(* CODESYS project untitled1.library
   Placeholder: TwinCAT_LIB
   Title: TwinCAT_LIB
   Version: 1.31
   Description: Baisc library's for s88 programming
   Company: Farnwood Engineering

Project tree, tasks and I/O mapping:
  libraries: Tc2_Standard, * (Beckhoff Automation GmbH); Tc2_System, * (Beckhoff Automation GmbH); Tc3_Module, * (Beckhoff Automation GmbH)
  DUTs/
  GVLs/
    POUs/
      LIB/
        1. Control Modules/
          1. DEV_Base/
            function block FB_DeviceBase [ST]
            data type stDevBase
          2. DEV_AnaIn/
            function block FB_DEV_AnaIn [ST]
            interface ITF_DEV_AnaIn
          3. DEV_DigIn/
            function block FB_DEV_DigIn [ST]: FB_init, Force, ResetForce, ActualValue, FallingEdge, RisingEdge
            interface ITF_DigIn: FB_init, Force, ResetForce, ActualValue, FallingEdge, RisingEdge
          4. DEV_Valve/
            ENUMs/
              data type E_ValveState
            STRUCTs/
              data type stDevValve
            function block DEV_Valve [ST]: _FExceptions, _StHmi, Close, Open, Reset, SetMode, ActualState, EmergencyStatus, OperatingMode
            interface ITF_Valve: Close, Open, Reset, SetMode, ActualState, EmergencyStatus, OperatingMode
          5. DEV_ControlValve/
            ENUMs/
              data type E_CtrlValveState
            STRUCTs/
            function block DEV_CtrlValve [ST]: EmergencyStatus, OperatingMode, OutputValue, Reset, SetMode, SetValue
            interface ITF_ControlValve: Reset, SetMode, SetValue, EmergencyStatus, OperatingMode, OutputValue
          6. DEV_Motor/
            ENUMs/
              data type E_MotorState
            STRUCTs/
            interface ITF_Motor: Auto, Manueel, Reset, Richting_L, Richting_R, Start, Stop, Toerental, ActualState, Error_State, State
          7. DEV_ControlMotor/
          ENUMs/
            data type E_OperationMode
          function block FB_Devices [ST]
        2. Equipment Modules/
          1. FB_Base/
            function block FB_EMbase [ST]
            data type stEMbase
          2. FB_Machine_PackML/
            data type E_State_PackML
            function block FB_Machine_PackML [ST]: Abort, Aborting_SC, Clear, Clearing_SC, Completing_SC, Execute_SC, Hold, Holding_SC, Reset, Resetting_SC, Start, Starting_SC, Stop, Stopping_SC, Suspend, Suspending_SC, Unhold, Unholding_SC, Unsuspend, Unsuspending_SC, State, FB_init
            interface ITF_PackML: Abort, Aborting_SC, Clear, Clearing_SC, Completing_SC, Execute_SC, Hold, Holding_SC, Reset, Resetting_SC, Start, Starting_SC, Stop, Stopping_SC, Suspend, Suspending_SC, Unhold, Unholding_SC, Unsuspend, Unsuspending_SC, State, FB_init
            data type STRUCT_fb_mem
          2. FB_Transport/
            data type E_Transport
            function block FB_Transport [ST]: Abort, Clear, Reset, Start, Stop, RPM, State, Tag
            interface ITF_FB_Transport: Abort, Clear, Reset, Start, Stop, RPM, State, Tag
            data type Str_FB_Transport
          3. FB_Transport_Mechanische_Stop/
            data type E_Mechanische_Stop
            function block FB_Mechanische_Stop [ST]: Close, Open, State, Tag
            interface ITF_FB_Transport_Mechanische_Stop: Close, Open, State, Tag
        3. Units/
          1. UN_Base/
            function block FB_UN_base [ST]
            data type stUNbase
        4. Management layer/
          FB_Alarmhandler/
      program MAIN [ST]
  Version/
    global variables Global_Version
  VISUs/
*)

// GVLs/POUs/LIB/1. Control Modules/1. DEV_Base/stDevBase
TYPE stDevBase :
STRUCT
	sTagName : STRING;
	sDescription : STRING;
END_STRUCT
END_TYPE

// GVLs/POUs/LIB/1. Control Modules/4. DEV_Valve/ENUMs/E_ValveState
{attribute 'qualified_only'}
{attribute 'strict'}
TYPE E_ValveState :
(
	Unknown := 0,
	Open := 1,
	Closed := 2,
	Opening := 3,
	Closing := 4,
	Error := -1
);
END_TYPE

// GVLs/POUs/LIB/1. Control Modules/4. DEV_Valve/STRUCTs/stDevValve
TYPE stDevValve :
STRUCT
	//Input to HMI
	bGetHmiError : BOOL;  //True = error
	bGetHmiStatus : BOOL; //True = Open || False = Closed
	eGetState : E_ValveState;
	eGetMode : E_OperationMode;
	
	//Output from HMI
	eSetMode : E_OperationMode; 
END_STRUCT
END_TYPE

// GVLs/POUs/LIB/1. Control Modules/5. DEV_ControlValve/ENUMs/E_CtrlValveState
{attribute 'qualified_only'}
{attribute 'strict'}
TYPE E_CtrlValveState :
(
	Unknown := 0,
	InPosition := 1,
	Moving := 2,
	Error := -1
);
END_TYPE

// GVLs/POUs/LIB/1. Control Modules/6. DEV_Motor/ENUMs/E_MotorState
{attribute 'qualified_only'}
{attribute 'strict'}
TYPE E_MotorState :
(
	Unknown := 0,
	Running := 1,
	Stalled := 2,
	SpeedingUp := 3,
	SpeedingDown := 4,
	Error := -1
);
END_TYPE

// GVLs/POUs/LIB/1. Control Modules/ENUMs/E_OperationMode
{attribute 'qualified_only'}
{attribute 'strict'}
TYPE E_OperationMode :
(
	Off := 0,
	Manual := 1,
	Automatic := 2
);
END_TYPE

// GVLs/POUs/LIB/2. Equipment Modules/1. FB_Base/stEMbase
TYPE stEMbase :
STRUCT
	sTagName : STRING;
	sDescription : STRING;
END_STRUCT
END_TYPE

// GVLs/POUs/LIB/2. Equipment Modules/2. FB_Machine_PackML/E_State_PackML
{attribute 'qualified_only'}
{attribute 'strict'}
TYPE E_State_PackML :
(
	IDLE	:= 0,
	STARTING,
	EXECUTE,
	COMPLETING,
	COMPLETE,
	RESETTING,
	HOLDING,
	HELD,
	UNHOLDING,
	SUSPENDING,
	SUSPENDED,
	UNSUSPENDING,
	ABORTING,
	ABORTED,
	CLEARING,
	STOPPING,
	STOPPED
);
END_TYPE

// GVLs/POUs/LIB/2. Equipment Modules/2. FB_Machine_PackML/STRUCT_fb_mem
TYPE STRUCT_fb_mem :
STRUCT
	//Properties
	State 			: E_State_PackML;
	//Methods
   	Abort 			: BOOL;
	Aborting_SC 	: BOOL;
	Clear 			: BOOL;
	Clearing_SC 	: BOOL;
	Execute_SC 		: BOOL;
	Completing_SC	: BOOL;
	Hold 			: BOOL;
	Holding_SC 		: BOOL;
	Reset 			: BOOL;
	Resetting_SC 	: BOOL;
	Start 			: BOOL;
	Starting_SC 	: BOOL;
	Stop 			: BOOL;
	Stopping_SC 	: BOOL;
	Suspend 		: BOOL;
	Suspending_SC 	: BOOL;
	Unhold 			: BOOL;
	Unholding_SC 	: BOOL;
	Unsuspend 		: BOOL;
	Unsuspending_SC : BOOL;
END_STRUCT
END_TYPE

// GVLs/POUs/LIB/2. Equipment Modules/2. FB_Transport/E_Transport
{attribute 'qualified_only'}
{attribute 'strict'}
TYPE E_Transport :
(
	IDLE := 0,
	STARTING,
	EXECUTE,
	STOPPING,
	STOPPED,
	ABORTING,
	ABORT,
	CLEARING,
	CLEARED,
	RESETTING
	
);
END_TYPE

// GVLs/POUs/LIB/2. Equipment Modules/2. FB_Transport/Str_FB_Transport
{attribute 'qualified_only'}
{attribute 'strict'}
TYPE Str_FB_Transport :
(
	enum_member := 0
);
END_TYPE

// GVLs/POUs/LIB/2. Equipment Modules/3. FB_Transport_Mechanische_Stop/E_Mechanische_Stop
{attribute 'qualified_only'}
{attribute 'strict'}
TYPE E_Mechanische_Stop :
(
	enum_member := 0
);
END_TYPE

// GVLs/POUs/LIB/3. Units/1. UN_Base/stUNbase
TYPE stUNbase :
STRUCT
	sTagName : STRING;
	sDescription : STRING;
END_STRUCT
END_TYPE

// Version/Global_Version
{attribute 'TcGenerated'}
{attribute 'no-analysis'}
{attribute 'linkalways'}
// This function has been automatically generated from the project information.
VAR_GLOBAL CONSTANT
	{attribute 'const_non_replaced'}
	stLibVersion_TwinCAT_LIB : ST_LibVersion := (iMajor := 1, iMinor := 31, iBuild := 0, iRevision := 0, nFlags := 1, sVersion := '1.31');
END_VAR

// GVLs/POUs/LIB/1. Control Modules/1. DEV_Base/FB_DeviceBase
FUNCTION_BLOCK FB_DeviceBase
VAR
	TagName : STRING;
	Description : STRING;
	TagID : INT;
END_VAR

END_FUNCTION_BLOCK

// GVLs/POUs/LIB/1. Control Modules/2. DEV_AnaIn/FB_DEV_AnaIn
FUNCTION_BLOCK FB_DEV_AnaIn EXTENDS FB_DeviceBase IMPLEMENTS ITF_DEV_AnaIn
VAR_INPUT
END_VAR
VAR_OUTPUT
END_VAR
VAR
END_VAR

END_FUNCTION_BLOCK

// GVLs/POUs/LIB/1. Control Modules/2. DEV_AnaIn/ITF_DEV_AnaIn
INTERFACE ITF_DEV_AnaIn

END_INTERFACE

// GVLs/POUs/LIB/1. Control Modules/3. DEV_DigIn/FB_DEV_DigIn
FUNCTION_BLOCK FB_DEV_DigIn EXTENDS FB_DeviceBase IMPLEMENTS ITF_DigIn
VAR
	
END_VAR

{warning 'add method implementation '}
METHOD FB_init : BOOL
VAR_INPUT
	(* if TRUE, the retain variables are initialized (warm start / cold start)*)
	bInitRetains	: BOOL;
	(* if TRUE, the instance afterwards gets moved into the copy code (online change)*)
	bInCopyCode	: BOOL;
END_VAR
END_METHOD

{warning 'add method implementation '}
METHOD Force : BOOL
VAR_INPUT
	ForceValue	: BOOL;
END_VAR
END_METHOD

{warning 'add method implementation '}
METHOD ResetForce : BOOL
END_METHOD

{warning 'add property implementation'}
PROPERTY ActualValue : BOOL
GET
END_GET
SET
END_SET
END_PROPERTY

{warning 'add property implementation'}
PROPERTY FallingEdge : BOOL
GET
END_GET
SET
END_SET
END_PROPERTY

{warning 'add property implementation'}
PROPERTY RisingEdge : BOOL
GET
END_GET
SET
END_SET
END_PROPERTY

END_FUNCTION_BLOCK

// GVLs/POUs/LIB/1. Control Modules/3. DEV_DigIn/ITF_DigIn
INTERFACE ITF_DigIn

METHOD FB_init : BOOL
VAR_INPUT
	bInitRetains : BOOL; // if TRUE, the retain variables are initialized (warm start / cold start)
	bInCopyCode : BOOL;  // if TRUE, the instance afterwards gets moved into the copy code (online change)
END_VAR
END_METHOD

METHOD Force : BOOL
VAR_INPUT
	ForceValue : BOOL;
END_VAR
END_METHOD

METHOD ResetForce : BOOL
VAR_INPUT
END_VAR
END_METHOD

PROPERTY ActualValue : BOOL
GET
END_GET
SET
END_SET
END_PROPERTY

PROPERTY FallingEdge : BOOL
GET
END_GET
SET
END_SET
END_PROPERTY

PROPERTY RisingEdge : BOOL
GET
END_GET
SET
END_SET
END_PROPERTY

END_INTERFACE

// GVLs/POUs/LIB/1. Control Modules/4. DEV_Valve/DEV_Valve
FUNCTION_BLOCK DEV_Valve EXTENDS FB_DeviceBase IMPLEMENTS ITF_Valve

VAR
	I_FeedbackOpen		AT	%I* : BOOL;
	I_FeedbackClosed 	AT 	%I* : BOOL;
	I_Estop				AT	%I*	: BOOL;
	Q_ValveOutput		AT	%Q*	: BOOL;
	
	s_eActualState				: E_ValveState;
	s_eOperatingMode			: E_OperationMode;
	s_tonFeedbackTime			: TON;
	
	bFeedbackError		: BOOL;
	bEstopActive		: BOOL;
	bBothFeedback		: BOOL;
END_VAR

METHOD _FExceptions : BOOL
VAR_INPUT
END_VAR
END_METHOD

METHOD PRIVATE _StHmi
VAR_INPUT
	stHMI : stDevValve;
END_VAR
END_METHOD

{warning 'add method implementation '}
METHOD Close : BOOL
END_METHOD

{warning 'add method implementation '}
METHOD Open : BOOL
END_METHOD

{warning 'add method implementation '}
METHOD Reset : BOOL
END_METHOD

{warning 'add method implementation '}
METHOD SetMode : BOOL
END_METHOD

{warning 'add property implementation'}
PROPERTY ActualState : E_ValveState
GET
END_GET
END_PROPERTY

{warning 'add property implementation'}
PROPERTY EmergencyStatus : BOOL
GET
END_GET
END_PROPERTY

{warning 'add property implementation'}
PROPERTY OperatingMode : BOOL
GET
END_GET
END_PROPERTY

END_FUNCTION_BLOCK

// GVLs/POUs/LIB/1. Control Modules/4. DEV_Valve/ITF_Valve
INTERFACE ITF_Valve

METHOD Close : BOOL
VAR_INPUT
END_VAR
END_METHOD

METHOD Open : BOOL
VAR_INPUT
END_VAR
END_METHOD

METHOD Reset : BOOL
VAR_INPUT
END_VAR
END_METHOD

METHOD SetMode : BOOL
VAR_INPUT
END_VAR
END_METHOD

PROPERTY ActualState : E_ValveState
GET
END_GET
END_PROPERTY

PROPERTY EmergencyStatus : BOOL
GET
END_GET
END_PROPERTY

PROPERTY OperatingMode : BOOL
GET
END_GET
END_PROPERTY

END_INTERFACE

// GVLs/POUs/LIB/1. Control Modules/5. DEV_ControlValve/DEV_CtrlValve
FUNCTION_BLOCK DEV_CtrlValve EXTENDS FB_DeviceBase IMPLEMENTS ITF_ControlValve
VAR_INPUT
END_VAR
VAR_OUTPUT
END_VAR
VAR
END_VAR

{warning 'add property implementation'}
PROPERTY EmergencyStatus : BOOL
GET
END_GET
END_PROPERTY

{warning 'add property implementation'}
PROPERTY OperatingMode : BOOL
GET
END_GET
END_PROPERTY

{warning 'add property implementation'}
PROPERTY OutputValue : REAL
GET
END_GET
END_PROPERTY

{warning 'add method implementation '}
METHOD Reset : BOOL
END_METHOD

{warning 'add method implementation '}
METHOD SetMode : BOOL
END_METHOD

{warning 'add method implementation '}
METHOD SetValue : BOOL
END_METHOD

END_FUNCTION_BLOCK

// GVLs/POUs/LIB/1. Control Modules/5. DEV_ControlValve/ITF_ControlValve
INTERFACE ITF_ControlValve

METHOD Reset : BOOL
VAR_INPUT
END_VAR
END_METHOD

METHOD SetMode : BOOL
VAR_INPUT
END_VAR
END_METHOD

METHOD SetValue : BOOL
VAR_INPUT
END_VAR
END_METHOD

PROPERTY EmergencyStatus : BOOL
GET
END_GET
END_PROPERTY

PROPERTY OperatingMode : BOOL
GET
END_GET
END_PROPERTY

PROPERTY OutputValue : REAL
GET
END_GET
END_PROPERTY

END_INTERFACE

// GVLs/POUs/LIB/1. Control Modules/6. DEV_Motor/ITF_Motor
INTERFACE ITF_Motor

METHOD Auto : BOOL
VAR_INPUT
END_VAR
END_METHOD

METHOD Manueel : BOOL
VAR_INPUT
END_VAR
END_METHOD

METHOD Reset : BOOL
VAR_INPUT
END_VAR
END_METHOD

METHOD Richting_L : BOOL
VAR_INPUT
END_VAR
END_METHOD

METHOD Richting_R : BOOL
VAR_INPUT
END_VAR
END_METHOD

METHOD Start : BOOL
VAR_INPUT
END_VAR
END_METHOD

METHOD Stop : BOOL
VAR_INPUT
END_VAR
END_METHOD

METHOD Toerental : INT
VAR_INPUT
END_VAR
END_METHOD

PROPERTY ActualState : BOOL
GET
END_GET
END_PROPERTY

PROPERTY Error_State : BOOL
GET
END_GET
END_PROPERTY

PROPERTY State : E_MotorState
GET
END_GET
END_PROPERTY

END_INTERFACE

// GVLs/POUs/LIB/1. Control Modules/FB_Devices
FUNCTION_BLOCK FB_Devices
VAR
	devValveV2012 : DEV_Valve := (TagName := 'V2012', Description := 'Standard Valve', TagID := 1);
	devValveV2020 : DEV_Valve := (TagName := 'V2020', Description := 'Standard Valve', TagID := 2);
	devValveV2021 : DEV_Valve := (TagName := 'V2021', Description := 'Standard Valve', TagID := 3);
	devValveV2022 : DEV_Valve := (TagName := 'V2022', Description := 'Standard Valve', TagID := 4);
END_VAR

devValveV2012();
devValveV2020();
devValveV2021();
devValveV2020();

END_FUNCTION_BLOCK

// GVLs/POUs/LIB/2. Equipment Modules/1. FB_Base/FB_EMbase
FUNCTION_BLOCK FB_EMbase
VAR
	TagName : STRING;
	Description : STRING;
	TagID : INT;
END_VAR

END_FUNCTION_BLOCK

// GVLs/POUs/LIB/2. Equipment Modules/2. FB_Machine_PackML/FB_Machine_PackML
FUNCTION_BLOCK FB_Machine_PackML IMPLEMENTS ITF_PackML
VAR
	fb_mem : STRUCT_fb_mem;
END_VAR

(*
$$$$$$$$\                                                                   $$\       $$$$$$$$\                     $$\                                         $$\                     
$$  _____|                                                                  $$ |      $$  _____|                    \__|                                        \__|                    
$$ |   $$$$$$\   $$$$$$\  $$$$$$$\  $$\  $$\  $$\  $$$$$$\   $$$$$$\   $$$$$$$ |      $$ |      $$$$$$$\   $$$$$$\  $$\ $$$$$$$\   $$$$$$\   $$$$$$\   $$$$$$\  $$\ $$$$$$$\   $$$$$$\  
$$$$$\ \____$$\ $$  __$$\ $$  __$$\ $$ | $$ | $$ |$$  __$$\ $$  __$$\ $$  __$$ |      $$$$$\    $$  __$$\ $$  __$$\ $$ |$$  __$$\ $$  __$$\ $$  __$$\ $$  __$$\ $$ |$$  __$$\ $$  __$$\ 
$$  __|$$$$$$$ |$$ |  \__|$$ |  $$ |$$ | $$ | $$ |$$ /  $$ |$$ /  $$ |$$ /  $$ |      $$  __|   $$ |  $$ |$$ /  $$ |$$ |$$ |  $$ |$$$$$$$$ |$$$$$$$$ |$$ |  \__|$$ |$$ |  $$ |$$ /  $$ |
$$ |  $$  __$$ |$$ |      $$ |  $$ |$$ | $$ | $$ |$$ |  $$ |$$ |  $$ |$$ |  $$ |      $$ |      $$ |  $$ |$$ |  $$ |$$ |$$ |  $$ |$$   ____|$$   ____|$$ |      $$ |$$ |  $$ |$$ |  $$ |
$$ |  \$$$$$$$ |$$ |      $$ |  $$ |\$$$$$\$$$$  |\$$$$$$  |\$$$$$$  |\$$$$$$$ |      $$$$$$$$\ $$ |  $$ |\$$$$$$$ |$$ |$$ |  $$ |\$$$$$$$\ \$$$$$$$\ $$ |      $$ |$$ |  $$ |\$$$$$$$ |
\__|   \_______|\__|      \__|  \__| \_____\____/  \______/  \______/  \_______|      \________|\__|  \__| \____$$ |\__|\__|  \__| \_______| \_______|\__|      \__|\__|  \__| \____$$ |
                                                                                                          $$\   $$ |                                                          $$\   $$ |
                                                                                                          \$$$$$$  |                                                          \$$$$$$  |
                                                                                                           \______/                                                            \______/ 
*)

CASE fb_mem.State OF
	E_State_PackML.IDLE 			: 
		//HAPPY FLOW		
		IF fb_mem.Start AND NOT fb_mem.Abort THEN
			fb_mem.State:= E_State_PackML.STARTING;
		END_IF
		
		//EXEPTION HANDLING
		IF fb_mem.Abort THEN
			fb_mem.State:= E_State_PackML.ABORTING;
		END_IF
		IF fb_mem.Stop THEN
			fb_mem.State:= E_State_PackML.STOPPING;
		END_IF
	
	E_State_PackML.STARTING 		:
		//HAPPY FLOW		
		IF fb_mem.Starting_SC AND NOT fb_mem.Abort THEN
			fb_mem.State:= E_State_PackML.IDLE;
		END_IF
		
		//EXEPTION HANDLING
		IF fb_mem.Abort THEN
			fb_mem.State:= E_State_PackML.ABORTING;
		END_IF
		IF fb_mem.Stop THEN
			fb_mem.State:= E_State_PackML.STOPPING;
		END_IF
	
	E_State_PackML.EXECUTE 			: 
		//HAPPY FLOW		
		IF fb_mem.Execute_SC AND NOT fb_mem.Abort THEN
			fb_mem.State:= E_State_PackML.IDLE;
		END_IF
		
		IF fb_mem.Hold THEN
			fb_mem.State:= E_State_PackML.HOLDING;
		END_IF
		
		IF fb_mem.Suspend THEN
			fb_mem.State:= E_State_PackML.SUSPENDED;
		END_IF
		
		//EXEPTION HANDLING
		IF fb_mem.Abort THEN
			fb_mem.State:= E_State_PackML.ABORTING;
		END_IF
		IF fb_mem.Stop THEN
			fb_mem.State:= E_State_PackML.STOPPING;
		END_IF
	
	E_State_PackML.COMPLETE 		:
		//HAPPY FLOW
		fb_mem.State:= E_State_PackML.RESETTING;
	
	E_State_PackML.RESETTING 		:
		//HAPPY FLOW		
		IF fb_mem.Resetting_SC AND NOT fb_mem.Abort THEN
			fb_mem.State:= E_State_PackML.IDLE;
		END_IF
		
		//EXEPTION HANDLING
		IF fb_mem.Abort THEN
			fb_mem.State:= E_State_PackML.ABORTING;
		END_IF
		IF fb_mem.Stop THEN
			fb_mem.State:= E_State_PackML.STOPPING;
		END_IF
	
	E_State_PackML.HOLDING 			:
		//HAPPY FLOW		
		IF fb_mem.Holding_SC AND NOT fb_mem.Abort THEN
			fb_mem.State:= E_State_PackML.HELD;
		END_IF
		
		//EXEPTION HANDLING
		IF fb_mem.Abort THEN
			fb_mem.State:= E_State_PackML.ABORTING;
		END_IF
		IF fb_mem.Stop THEN
			fb_mem.State:= E_State_PackML.STOPPING;
		END_IF
		
	
	E_State_PackML.HELD 			:
		//HAPPY FLOW		
		IF fb_mem.Unhold AND NOT fb_mem.Abort THEN
			fb_mem.State:= E_State_PackML.UNHOLDING;
		END_IF
		
		//EXEPTION HANDLING
		IF fb_mem.Abort THEN
			fb_mem.State:= E_State_PackML.ABORTING;
		END_IF
		IF fb_mem.Stop THEN
			fb_mem.State:= E_State_PackML.STOPPING;
		END_IF
	
	E_State_PackML.UNHOLDING 		:
		//HAPPY FLOW		
		IF fb_mem.Unholding_SC AND NOT fb_mem.Abort THEN
			fb_mem.State:= E_State_PackML.EXECUTE;
		END_IF
		
		//EXEPTION HANDLING
		IF fb_mem.Abort THEN
			fb_mem.State:= E_State_PackML.ABORTING;
		END_IF
		IF fb_mem.Stop THEN
			fb_mem.State:= E_State_PackML.STOPPING;
		END_IF
	
	E_State_PackML.SUSPENDING 		:
		//HAPPY FLOW		
		IF fb_mem.Suspending_SC AND NOT fb_mem.Abort THEN
			fb_mem.State:= E_State_PackML.SUSPENDED;
		END_IF
		
		//EXEPTION HANDLING
		IF fb_mem.Abort THEN
			fb_mem.State:= E_State_PackML.ABORTING;
		END_IF
		IF fb_mem.Stop THEN
			fb_mem.State:= E_State_PackML.STOPPING;
		END_IF
	
	
	E_State_PackML.SUSPENDED 		:
		//HAPPY FLOW		
		IF fb_mem.Unsuspend AND NOT fb_mem.Abort THEN
			fb_mem.State:= E_State_PackML.UNSUSPENDING;
		END_IF
		
		//EXEPTION HANDLING
		IF fb_mem.Abort THEN
			fb_mem.State:= E_State_PackML.ABORTING;
		END_IF
		IF fb_mem.Stop THEN
			fb_mem.State:= E_State_PackML.STOPPING;
		END_IF
	
	E_State_PackML.UNSUSPENDING 	:
		//HAPPY FLOW		
		IF fb_mem.Unsuspending_SC AND NOT fb_mem.Abort THEN
			fb_mem.State:= E_State_PackML.EXECUTE;
		END_IF
		
		//EXEPTION HANDLING
		IF fb_mem.Abort THEN
			fb_mem.State:= E_State_PackML.ABORTING;
		END_IF
		IF fb_mem.Stop THEN
			fb_mem.State:= E_State_PackML.STOPPING;
		END_IF
	
	E_State_PackML.ABORTED			:
		//HAPPY FLOW		
		IF fb_mem.Clear THEN
			fb_mem.State:= E_State_PackML.CLEARING;
		END_IF
	
		
	E_State_PackML.ABORTING			:
		//HAPPY FLOW		
		IF fb_mem.Aborting_SC THEN
			fb_mem.State:= E_State_PackML.ABORTED;
		END_IF
	
		
	E_State_PackML.CLEARING 		:
		//HAPPY FLOW		
		IF fb_mem.Clearing_SC THEN
			fb_mem.State:= E_State_PackML.STOPPED;
		END_IF
		
		//EXEPTION HANDLING
		IF fb_mem.Abort THEN
			fb_mem.State:= E_State_PackML.ABORTING;
		END_IF
		
		
	E_State_PackML.STOPPING 		:
		//HAPPY FLOW
		IF fb_mem.Stopping_SC THEN
			fb_mem.State:= E_State_PackML.STOPPED;
		END_IF
		
		//EXEPTION HANDLING
		IF fb_mem.Abort THEN
			fb_mem.State:= E_State_PackML.ABORTING;
		END_IF
		
	
	E_State_PackML.STOPPED 			: 
		//HAPPY FLOW
		IF fb_mem.Reset AND NOT fb_mem.Abort THEN
			fb_mem.State:= E_State_PackML.RESETTING;
		END_IF
		
		//EXEPTION HANDLING
		IF fb_mem.Abort THEN
			fb_mem.State:= E_State_PackML.ABORTING;
		END_IF
		IF fb_mem.Stop THEN
			fb_mem.State:= E_State_PackML.STOPPING;
		END_IF
END_CASE

{warning 'add method implementation '}
METHOD Abort : BOOL
fb_mem.Abort := TRUE;
END_METHOD

{warning 'add method implementation '}
METHOD Aborting_SC : BOOL
fb_mem.Aborting_SC := TRUE;
END_METHOD

{warning 'add method implementation '}
METHOD Clear : BOOL
fb_mem.Clear := TRUE;
END_METHOD

{warning 'add method implementation '}
METHOD Clearing_SC : BOOL
fb_mem.Clearing_SC := TRUE;
END_METHOD

{warning 'add method implementation '}
METHOD Completing_SC : BOOL
fb_mem.Completing_SC := TRUE;
END_METHOD

{warning 'add method implementation '}
METHOD Execute_SC : BOOL
fb_mem.Execute_SC := TRUE;
END_METHOD

{warning 'add method implementation '}
METHOD Hold : BOOL
fb_mem.Hold := TRUE;
END_METHOD

{warning 'add method implementation '}
METHOD Holding_SC : BOOL
fb_mem.Holding_SC := TRUE;
END_METHOD

{warning 'add method implementation '}
METHOD Reset : BOOL
fb_mem.Reset := TRUE;
END_METHOD

{warning 'add method implementation '}
METHOD Resetting_SC : BOOL
fb_mem.Resetting_SC := TRUE;
END_METHOD

{warning 'add method implementation '}
METHOD Start : BOOL
fb_mem.Start := TRUE;
END_METHOD

{warning 'add method implementation '}
METHOD Starting_SC : BOOL
fb_mem.Starting_SC := TRUE;
END_METHOD

{warning 'add method implementation '}
METHOD Stop : BOOL
fb_mem.Stop := TRUE;
END_METHOD

{warning 'add method implementation '}
METHOD Stopping_SC : BOOL
fb_mem.Stopping_SC := TRUE;
END_METHOD

{warning 'add method implementation '}
METHOD Suspend : BOOL
fb_mem.Suspend := TRUE;
END_METHOD

{warning 'add method implementation '}
METHOD Suspending_SC : BOOL
fb_mem.Suspending_SC := TRUE;
END_METHOD

{warning 'add method implementation '}
METHOD Unhold : BOOL
fb_mem.Unhold := TRUE;
END_METHOD

{warning 'add method implementation '}
METHOD Unholding_SC : BOOL
fb_mem.Unholding_SC := TRUE;
END_METHOD

{warning 'add method implementation '}
METHOD Unsuspend : BOOL
fb_mem.Unsuspend := TRUE;
END_METHOD

METHOD Unsuspending_SC : BOOL
VAR_INPUT
END_VAR
fb_mem.Unsuspending_SC := TRUE;
END_METHOD

{warning 'add property implementation'}
PROPERTY State : E_State_PackML
GET
State := fb_mem.State;
END_GET
END_PROPERTY

METHOD FB_init : BOOL
VAR_INPUT
    bInitRetains : BOOL; // if TRUE, the retain variables are initialized (warm start / cold start)
    bInCopyCode  : BOOL; // if TRUE, the instance afterwards gets moved into the copy code (online change)
END_VAR
END_METHOD

END_FUNCTION_BLOCK

// GVLs/POUs/LIB/2. Equipment Modules/2. FB_Machine_PackML/ITF_PackML
INTERFACE ITF_PackML

METHOD Abort : BOOL
VAR_INPUT
END_VAR
END_METHOD

METHOD Aborting_SC : BOOL
VAR_INPUT
END_VAR
END_METHOD

METHOD Clear : BOOL
VAR_INPUT
END_VAR
END_METHOD

METHOD Clearing_SC : BOOL
VAR_INPUT
END_VAR
END_METHOD

METHOD Completing_SC : BOOL
VAR_INPUT
END_VAR
END_METHOD

METHOD Execute_SC : BOOL
VAR_INPUT
END_VAR
END_METHOD

METHOD Hold : BOOL
VAR_INPUT
END_VAR
END_METHOD

METHOD Holding_SC : BOOL
VAR_INPUT
END_VAR
END_METHOD

METHOD Reset : BOOL
VAR_INPUT
END_VAR
END_METHOD

METHOD Resetting_SC : BOOL
VAR_INPUT
END_VAR
END_METHOD

METHOD Start : BOOL
VAR_INPUT
END_VAR
END_METHOD

METHOD Starting_SC : BOOL
VAR_INPUT
END_VAR
END_METHOD

METHOD Stop : BOOL
VAR_INPUT
END_VAR
END_METHOD

METHOD Stopping_SC : BOOL
VAR_INPUT
END_VAR
END_METHOD

METHOD Suspend : BOOL
VAR_INPUT
END_VAR
END_METHOD

METHOD Suspending_SC : BOOL
VAR_INPUT
END_VAR
END_METHOD

METHOD Unhold : BOOL
VAR_INPUT
END_VAR
END_METHOD

METHOD Unholding_SC : BOOL
VAR_INPUT
END_VAR
END_METHOD

METHOD Unsuspend : BOOL
VAR_INPUT
END_VAR
END_METHOD

METHOD Unsuspending_SC : BOOL
VAR_INPUT
END_VAR
END_METHOD

PROPERTY State : E_State_PackML
GET
END_GET
END_PROPERTY

METHOD FB_init : BOOL
VAR_INPUT
	bInitRetains : BOOL; // if TRUE, the retain variables are initialized (warm start / cold start)
	bInCopyCode : BOOL;  // if TRUE, the instance afterwards gets moved into the copy code (online change)
END_VAR
END_METHOD

END_INTERFACE

// GVLs/POUs/LIB/2. Equipment Modules/2. FB_Transport/FB_Transport
FUNCTION_BLOCK FB_Transport IMPLEMENTS  ITF_FB_Transport

VAR
	fb_mem : Str_FB_Transport;
END_VAR

{warning 'add method implementation '}
METHOD Abort : BOOL
END_METHOD

{warning 'add method implementation '}
METHOD Clear : BOOL
END_METHOD

{warning 'add method implementation '}
METHOD Reset : BOOL
END_METHOD

{warning 'add method implementation '}
METHOD Start : BOOL
END_METHOD

{warning 'add method implementation '}
METHOD Stop : BOOL
END_METHOD

{warning 'add property implementation'}
PROPERTY RPM : INT
GET
END_GET
SET
END_SET
END_PROPERTY

{warning 'add property implementation'}
PROPERTY State : E_Transport
GET
END_GET
END_PROPERTY

{warning 'add property implementation'}
PROPERTY Tag : STRING
GET
END_GET
END_PROPERTY

END_FUNCTION_BLOCK

// GVLs/POUs/LIB/2. Equipment Modules/2. FB_Transport/ITF_FB_Transport
INTERFACE ITF_FB_Transport

METHOD Abort : BOOL
VAR_INPUT
END_VAR
END_METHOD

METHOD Clear : BOOL
VAR_INPUT
END_VAR
END_METHOD

METHOD Reset : BOOL
VAR_INPUT
END_VAR
END_METHOD

METHOD Start : BOOL
VAR_INPUT
END_VAR
END_METHOD

METHOD Stop : BOOL
VAR_INPUT
END_VAR
END_METHOD

PROPERTY RPM : INT
GET
END_GET
SET
END_SET
END_PROPERTY

PROPERTY State : E_Transport
GET
END_GET
END_PROPERTY

PROPERTY Tag : STRING
GET
END_GET
END_PROPERTY

END_INTERFACE

// GVLs/POUs/LIB/2. Equipment Modules/3. FB_Transport_Mechanische_Stop/FB_Mechanische_Stop
FUNCTION_BLOCK FB_Mechanische_Stop IMPLEMENTS  ITF_FB_Transport_Mechanische_Stop

VAR
END_VAR

{warning 'add method implementation '}
METHOD Close : BOOL
END_METHOD

{warning 'add method implementation '}
METHOD Open : BOOL
END_METHOD

{warning 'add property implementation'}
PROPERTY State : E_Mechanische_Stop
GET
END_GET
END_PROPERTY

{warning 'add property implementation'}
PROPERTY Tag : STRING
GET
END_GET
END_PROPERTY

END_FUNCTION_BLOCK

// GVLs/POUs/LIB/2. Equipment Modules/3. FB_Transport_Mechanische_Stop/ITF_FB_Transport_Mechanische_Stop
INTERFACE ITF_FB_Transport_Mechanische_Stop

METHOD Close : BOOL
VAR_INPUT
END_VAR
END_METHOD

METHOD Open : BOOL
VAR_INPUT
END_VAR
END_METHOD

PROPERTY State : E_Mechanische_Stop
GET
END_GET
END_PROPERTY

PROPERTY Tag : INT
GET
END_GET
END_PROPERTY

END_INTERFACE

// GVLs/POUs/LIB/3. Units/1. UN_Base/FB_UN_base
FUNCTION_BLOCK FB_UN_base
VAR
	TagName : STRING;
	Description : STRING;
	TagID : INT;
END_VAR

END_FUNCTION_BLOCK

// GVLs/POUs/MAIN
PROGRAM MAIN
VAR
END_VAR

END_PROGRAM
